TYPE ST_DataStuff :

STRUCT
	nFunctionID : UDINT;
	nRecordedValue : UDINT;	
END_STRUCT

END_TYPE

(* stored: Version 1.1.0.1, ProductVersion 3.1.4024.12
   DUT ST_DataStuff: Id {41474842-2cd0-42c5-a7f9-a3a7c94c5abb} *)
